PROGRAM MAIN
VAR



	SGO: TOGGLE;
	SGC: TOGGLE;
	TRU: TOGGLE;
	TRD: TOGGLE;
	VS: TOGGLE;
	TFS: TOGGLE;
	HSC: TOGGLE;
	HSO: TOGGLE;
	HDO: TOGGLE;
	HDC: TOGGLE;
	LC: TOGGLE;
	LR: TOGGLE;


	Eject_Empty_Pallet: BOOL;
	Empty_Pallet_Ejecting: BOOL;
	Empty_Pallet: BOOL;
	Full_Pallet: BOOL;
	Shroud_Latch: BOOL;


	Hoist_Cycle: BOOL;
	Next_Tier: BOOL;
	Hoist_Up_Disable: BOOL;
	ChainHoist_Enable: BOOL;
	Rev_Enable: BOOL;

	Auto_Tog: TOGGLE;



	Delay_Pallet_Advance2: TON;

	Delay_Pallet_Advance: TON;
	sChamberChain_Run: BOOL;
	Hoist_Down_Complete_TMR: TON;
	Discharge1_Pallet: BOOL;
	Eject_Cycle_TMR: TON;
	Hoist_Up_Tog: TOGGLE;
	Height_TMR: TOF;
	Reset_One_Shot: TP;
	sHoistUpDisable: BOOL;
	sChainHoistDn: BOOL;
	Fwd_Delay: TON;
	sCarriage_to_Pickup: BOOL;

	Open_Delay: TON;

	Release_Capture: TOF;
	DR2_Tog: TOGGLE;
	DR3_Tog: TOGGLE;
	DR4_Tog: TOGGLE;
	HoistUpDisableTog: TOGGLE;
	Gate_Closure_TMR:TON;




	Pa1Tog: TOGGLE;
	OpenTMR: TOF;
	CloseTMR: TOF;
	Down_Slow_Delay: TON;
	DSD: TIME;
	test: BOOL;
	Last_TierTMR1: TOF;
	Last_TierTMR2: TON;

	Down_Completion_TMR: TOF;
	Maintainloading: TOF;
	Ejecting_Pallet: BOOL;
	EmptyPallet_Jam_TMR: TON;





	TopFrameRem: TOF;
	Hoist_OneShot: TP;
	Hoist_Dn_Fast_Limit: TON;
	HDFL: TIME;
	Carriage_Disable_For_New_Pallet: BOOL;
	Slow_Reset: TP;
	LCT_Maintain: TOF;
	TT_Maintain: TOF;
	Disch1_Maintain: TOF;
	Disch2_Maintain: TOF;



	AutoLoadingTog: TOGGLE;
	ManualLoadingTog: TOGGLE;

	StopHoist_Tog: TOGGLE;

	TableTopJam: TON;
	Disch2Delay: TON;

	Discharge2Jam: TON;


	Disch2Full: TON;
	DR3TP: TP;
	Discharge2TOG: TOGGLE;
	Can_Count_M2: CTU;
	CC2: REAL;
	CanCount2A: CTU;
	CanCount2B: CTU;
	CC2B: REAL;
	CanCntReset: BOOL;
	CC2_Tens: REAL;

	FwdMaintain: TOF;
	Top_Frame_Removal: TON;
	Carriage_Forward_Enable: BOOL;
	Close_Pulse: TP;
	TT_Jam_Manager: TOF;
	Reverse_Delay: TON;
	Flash1_NP: TON;
	Flash2_NP: TOF;


	Flash1B: TON;
	Flash2B: TOF;
	mt: TOF;
	SlowTest: BOOL;
	Down_Slow_Maintain: TOF;
	Last_Slip_Sheet: TON;
	Test1: BOOL;
	Test2: BOOL;
	Empty_Pallet_Pulse: TP;
	Clank2_TMR: TON;
	Discharge_Run_TMR: TOF;
	Carriage_Slow_Enable: BOOL;
	Slow_Maintain: TOF;
	sc_DepalM2Count: INT;
	M2CanCounter2: CTU;
	M2CanCounter3: CTU;
	sc_Depal2Count3: BOOL;
	sc_Depal2Count2: BOOL;
	sc_Depal2Count13: INT;
	sc_Depal2Count12: INT;
	M2CanCounter4: CTU;
	M2CanCounter33: CTU;
	M2CanCounter34: CTU;
	a: INT;
	b: INT;
	C: INT;
	M2CanCounter333: CTU;
	d: INT;
	e: INT;
	F: INT;
	M2CanCounter333333: CTU;
	M: INT;
	DFS: CTU;
	LINCOLN: BOOL;

	LDS: BOOL;
	DSS: BOOL;
	K: INT;
	KJSJHE: BOOL;
	PLOP: INT;
	HLJKLTFK: CTU;
	FGHJD: INT;
	CancounterM2: CTU;
	CancounterM12: CTU;
	sc_Depal1_1stshiftcount: INT;
	try: INT;
	COUNTPULSE: BOOL;
	_TEST: CTU;
	_1stshiftcc: INT;
	_2NDshiftcc: INT;
	sc_M1CCReset: BOOL;
	Pallet_Count: INT;
	EmptyCans_Initial: REAL;
	InitialPalletCount: INT:=3276;
	TESTPALLETCOUNT: CTU;
	TESTPC: INT;
	M2CanCNTPE: BOOL;
	M2CanCountPE: BOOL;
	CanCounterCTU: CTU;
	CanCountWORD: WORD;
	CanCountMultiplier: CTU;
	MultiplierWORD: WORD;
	HighCount: REAL;
	MultiplierREAL: REAL;
	CanCountREAL: REAL;
	ActualCount: REAL;
	ChainHoistDown: Toggle;
	CHainHoistUp: TOGGLE;
	Infeed1: TOGGLE;
	ElevatorInfeed: TOGGLE;
	Elevatorrev: TOGGLE;
	Infeed2: Toggle;
	Infeed2REV: Toggle;
	Infeed1REV: TOGGLE;
	ELETOggle: TOGGLE;
	Cap: TOGGLE;
	Capture: TOGGLE;
	Release: TOGGLE;
	Rel: TOGGLE;
	hsclose: TOGGLE;
	sHoistSClose: BOOL;
	ABCD: TOGGLE;
	efgh: TOGGLE;
	CarFwd: Toggle;
	CarRev: Toggle;
	sDischarge1Run: BOOL;
	Discharge1Toggle: Toggle;
	Discharge2Run: Toggle;
	sDischarge2Run: BOOL;
	GD1: BOOL;
	Verify: TON;
	SetForNewPallet: SR;
	SendCarriageBack: BOOL;
	SetCarrRev: BOOL;
	Hoist_Tog_Resets: BOOL;
END_VAR
VAR_INPUT
	ProductHeight_Pos: BOOL;
	Carriage_to_Pickup: BOOL;
	Fwd_Enable: BOOL;
	DR1_Tog: TOGGLE;


END_VAR
VAR // added by the converter: edge detectors and wires of the graphical bodies
    _w1, _w2, _w3, _w4, _w5, _w6, _w7, _w8 : BOOL;
END_VAR

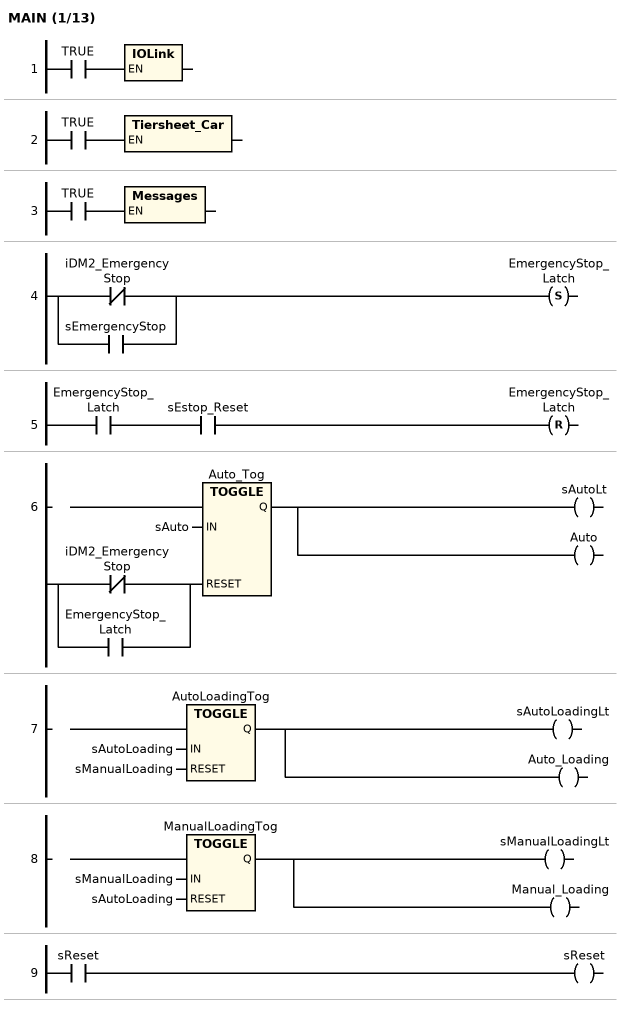
// NETWORK 1
IOLink();

// NETWORK 2
Tiersheet_Car();

// NETWORK 3
Messages();

// NETWORK 4
EmergencyStop_Latch S= NOT iDM2_EmergencyStop OR sEmergencyStop;

// NETWORK 5
EmergencyStop_Latch R= EmergencyStop_Latch AND sEstop_Reset;

// NETWORK 6
Auto_Tog(IN := sAuto, RESET := NOT iDM2_EmergencyStop OR EmergencyStop_Latch); // TOGGLE
sAutoLt := Auto_Tog.Q;
Auto := Auto_Tog.Q;

// NETWORK 7
AutoLoadingTog(IN := sAutoLoading, RESET := sManualLoading); // TOGGLE
sAutoLoadingLt := AutoLoadingTog.Q;
Auto_Loading := AutoLoadingTog.Q;

// NETWORK 8
ManualLoadingTog(IN := sManualLoading, RESET := sAutoLoading); // TOGGLE
sManualLoadingLt := ManualLoadingTog.Q;
Manual_Loading := ManualLoadingTog.Q;

// NETWORK 9
sReset := sReset;

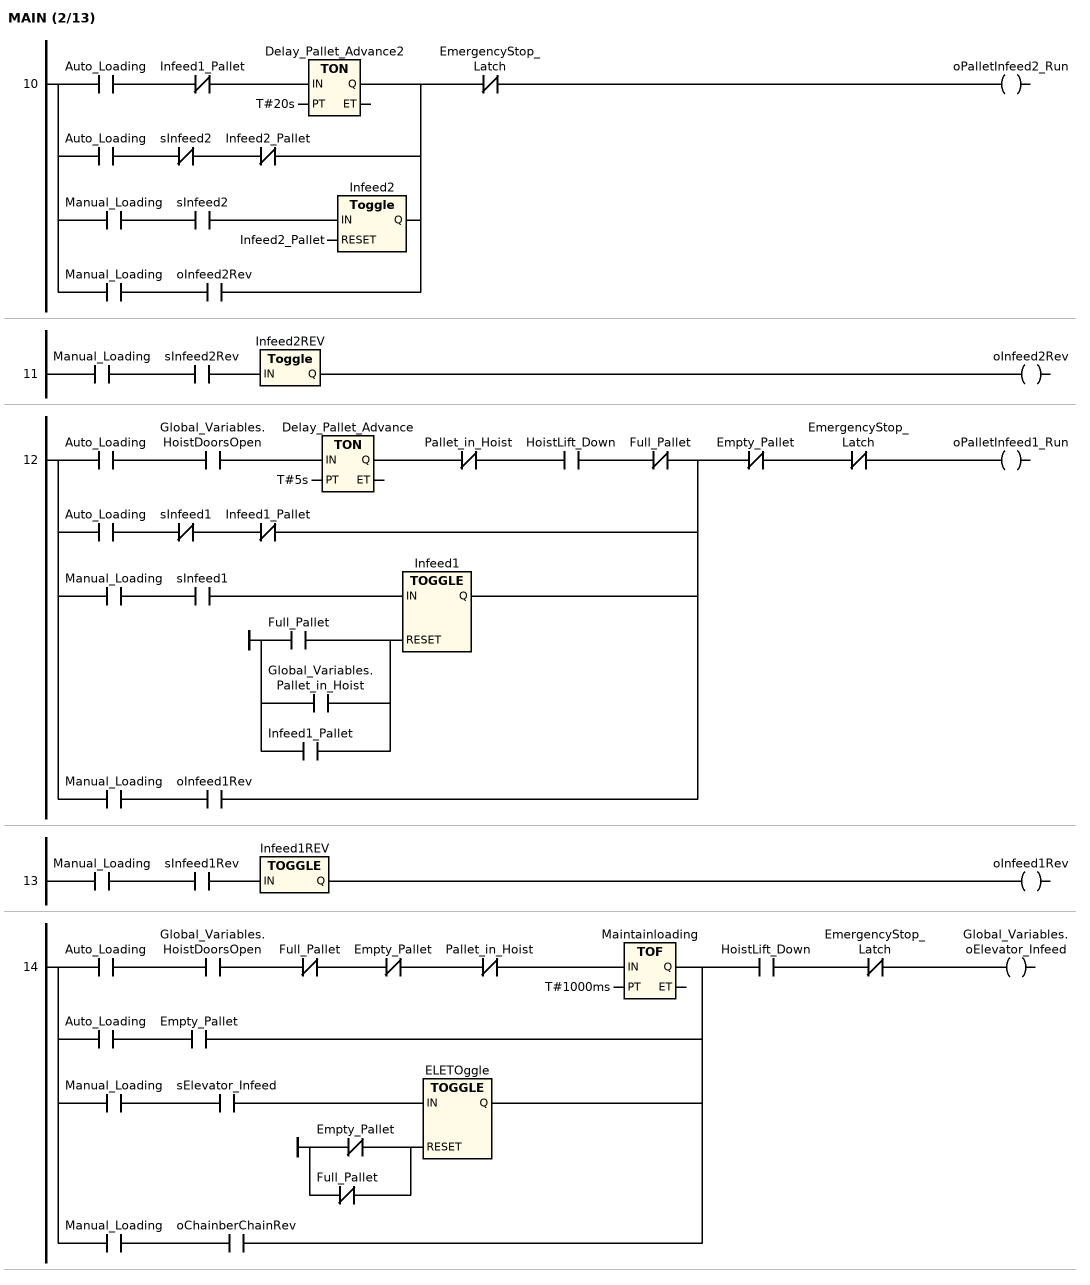
// NETWORK 10
Delay_Pallet_Advance2(IN := Auto_Loading AND NOT Infeed1_Pallet, PT := T#20s); // TON
Infeed2(IN := Manual_Loading AND sInfeed2, RESET := Infeed2_Pallet); // Toggle
oPalletInfeed2_Run := (Delay_Pallet_Advance2.Q OR Auto_Loading AND NOT sInfeed2 AND NOT Infeed2_Pallet OR Infeed2.Q OR Manual_Loading AND oInfeed2Rev) AND NOT EmergencyStop_Latch;

// NETWORK 11
Infeed2REV(IN := Manual_Loading AND sInfeed2Rev); // Toggle
oInfeed2Rev := Infeed2REV.Q;

// NETWORK 12
Delay_Pallet_Advance(IN := Auto_Loading AND Global_Variables.HoistDoorsOpen, PT := T#5s); // TON
Infeed1(IN := Manual_Loading AND sInfeed1, RESET := Full_Pallet OR Global_Variables.Pallet_in_Hoist OR Infeed1_Pallet); // TOGGLE
oPalletInfeed1_Run := (Delay_Pallet_Advance.Q AND NOT Pallet_in_Hoist AND HoistLift_Down AND NOT Full_Pallet OR Auto_Loading AND NOT sInfeed1 AND NOT Infeed1_Pallet OR Infeed1.Q OR Manual_Loading AND oInfeed1Rev) AND NOT Empty_Pallet AND NOT EmergencyStop_Latch;

// NETWORK 13
Infeed1REV(IN := Manual_Loading AND sInfeed1Rev); // TOGGLE
oInfeed1Rev := Infeed1REV.Q;

// NETWORK 14
Maintainloading(IN := Auto_Loading AND Global_Variables.HoistDoorsOpen AND NOT Full_Pallet AND NOT Empty_Pallet AND NOT Pallet_in_Hoist, PT := T#1000ms); // TOF
ELETOggle(IN := Manual_Loading AND sElevator_Infeed, RESET := NOT Empty_Pallet OR NOT Full_Pallet); // TOGGLE
Global_Variables.oElevator_Infeed := (Maintainloading.Q OR Auto_Loading AND Empty_Pallet OR ELETOggle.Q OR Manual_Loading AND oChainberChainRev) AND HoistLift_Down AND NOT EmergencyStop_Latch;

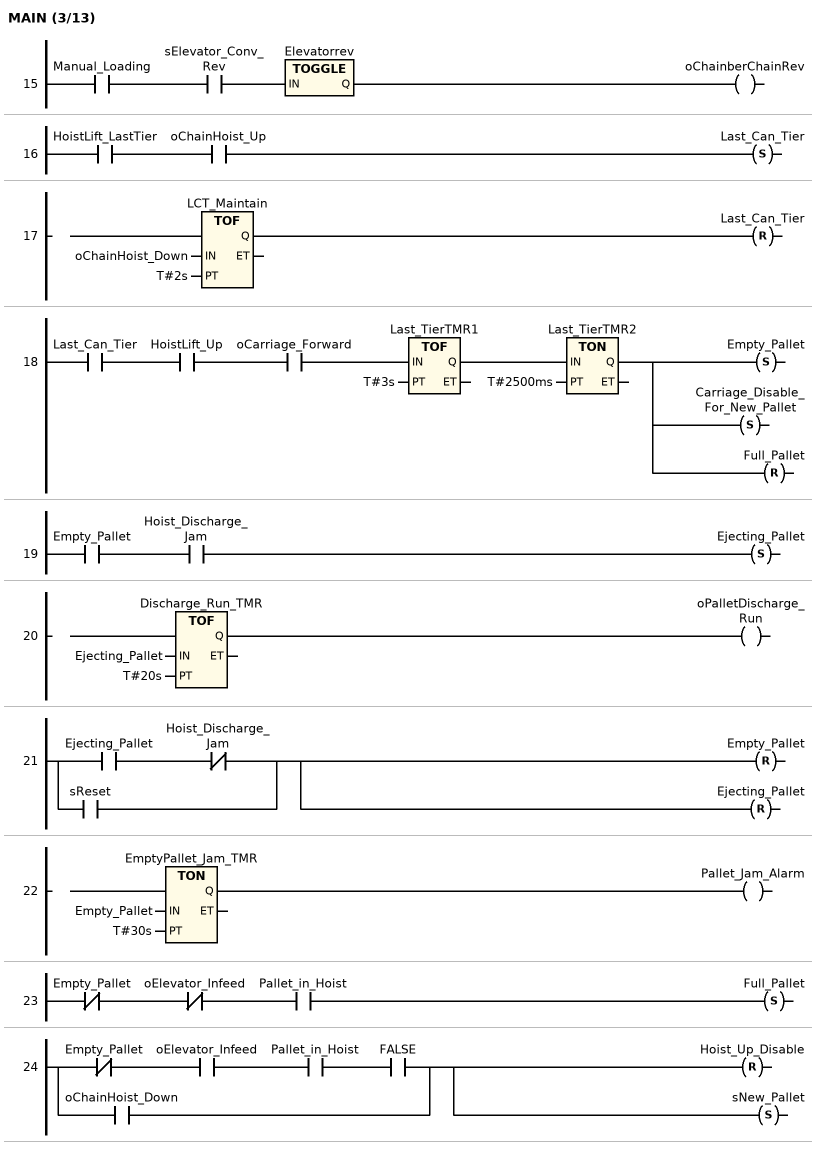
// NETWORK 15
Elevatorrev(IN := Manual_Loading AND sElevator_Conv_Rev); // TOGGLE
oChainberChainRev := Elevatorrev.Q;

// NETWORK 16
Last_Can_Tier S= HoistLift_LastTier AND oChainHoist_Up;

// NETWORK 17
LCT_Maintain(IN := oChainHoist_Down, PT := T#2s); // TOF
Last_Can_Tier R= LCT_Maintain.Q;

// NETWORK 18
Last_TierTMR1(IN := Last_Can_Tier AND HoistLift_Up AND oCarriage_Forward, PT := T#3s); // TOF
Last_TierTMR2(IN := Last_TierTMR1.Q, PT := T#2500ms); // TON
Empty_Pallet S= Last_TierTMR2.Q;
Carriage_Disable_For_New_Pallet S= Last_TierTMR2.Q;
Full_Pallet R= Last_TierTMR2.Q;

// NETWORK 19
Ejecting_Pallet S= Empty_Pallet AND Hoist_Discharge_Jam;

// NETWORK 20
Discharge_Run_TMR(IN := Ejecting_Pallet, PT := T#20s); // TOF
oPalletDischarge_Run := Discharge_Run_TMR.Q;

// NETWORK 21
_w1 := Ejecting_Pallet AND NOT Hoist_Discharge_Jam OR sReset;
Empty_Pallet R= _w1;
Ejecting_Pallet R= _w1;

// NETWORK 22
EmptyPallet_Jam_TMR(IN := Empty_Pallet, PT := T#30s); // TON
Pallet_Jam_Alarm := EmptyPallet_Jam_TMR.Q;

// NETWORK 23
Full_Pallet S= NOT Empty_Pallet AND NOT oElevator_Infeed AND Pallet_in_Hoist;

// NETWORK 24
_w2 := NOT Empty_Pallet AND oElevator_Infeed AND Pallet_in_Hoist AND FALSE OR oChainHoist_Down;
Hoist_Up_Disable R= _w2;
sNew_Pallet S= _w2;

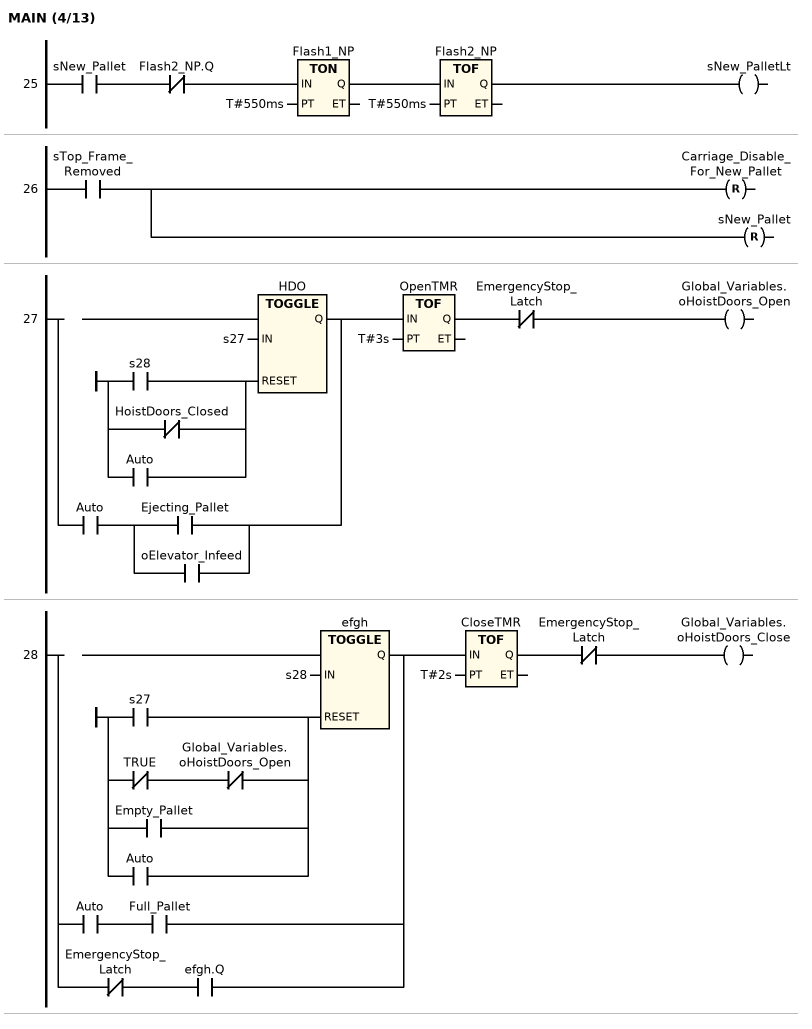
// NETWORK 25
Flash1_NP(IN := sNew_Pallet AND NOT Flash2_NP.Q, PT := T#550ms); // TON
Flash2_NP(IN := Flash1_NP.Q, PT := T#550ms); // TOF
sNew_PalletLt := Flash2_NP.Q;

// NETWORK 26
Carriage_Disable_For_New_Pallet R= sTop_Frame_Removed;
sNew_Pallet R= sTop_Frame_Removed;

// NETWORK 27
HDO(IN := s27, RESET := s28 OR NOT HoistDoors_Closed OR Auto); // TOGGLE
OpenTMR(IN := HDO.Q OR Auto AND (Ejecting_Pallet OR oElevator_Infeed), PT := T#3s); // TOF
Global_Variables.oHoistDoors_Open := OpenTMR.Q AND NOT EmergencyStop_Latch;

// NETWORK 28
efgh(IN := s28, RESET := s27 OR NOT TRUE AND NOT Global_Variables.oHoistDoors_Open OR Empty_Pallet OR Auto); // TOGGLE
CloseTMR(IN := efgh.Q OR Auto AND Full_Pallet OR NOT EmergencyStop_Latch AND efgh.Q, PT := T#2s); // TOF
Global_Variables.oHoistDoors_Close := CloseTMR.Q AND NOT EmergencyStop_Latch;

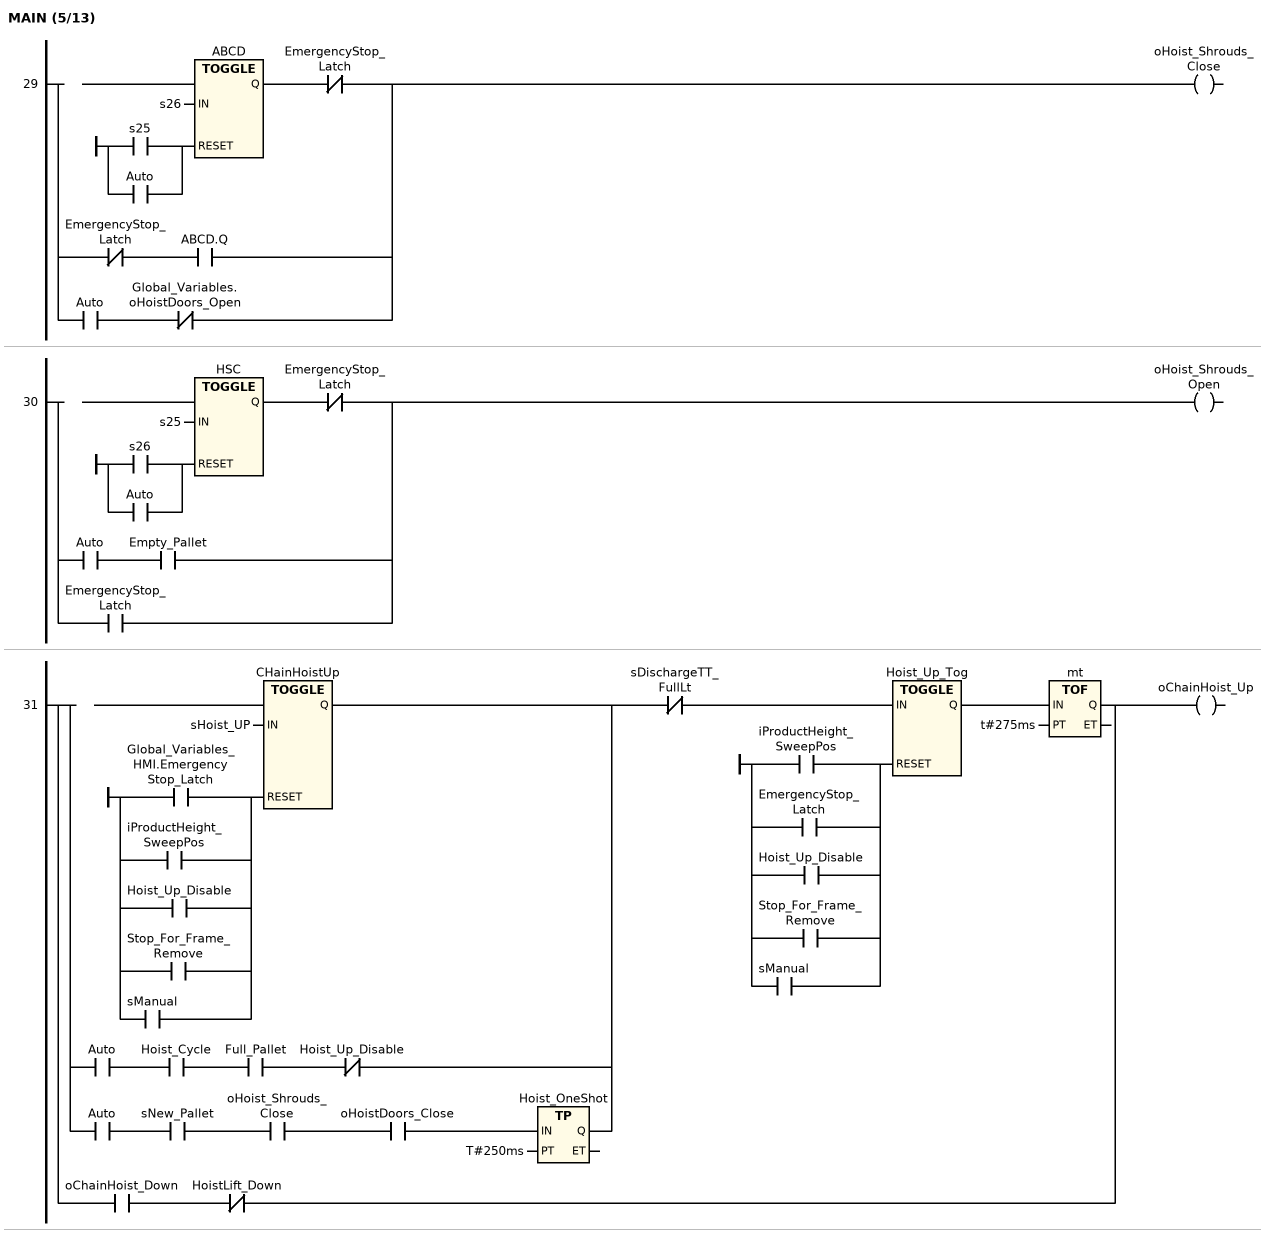
// NETWORK 29
ABCD(IN := s26, RESET := s25 OR Auto); // TOGGLE
oHoist_Shrouds_Close := ABCD.Q AND NOT EmergencyStop_Latch OR NOT EmergencyStop_Latch AND ABCD.Q OR Auto AND NOT Global_Variables.oHoistDoors_Open;

// NETWORK 30
HSC(IN := s25, RESET := s26 OR Auto); // TOGGLE
oHoist_Shrouds_Open := HSC.Q AND NOT EmergencyStop_Latch OR Auto AND Empty_Pallet OR EmergencyStop_Latch;

// NETWORK 31
CHainHoistUp(IN := sHoist_UP, RESET := Global_Variables_HMI.EmergencyStop_Latch OR iProductHeight_SweepPos OR Hoist_Up_Disable OR Stop_For_Frame_Remove OR sManual); // TOGGLE
Hoist_OneShot(IN := Auto AND sNew_Pallet AND oHoist_Shrouds_Close AND oHoistDoors_Close, PT := T#250ms); // TP
Hoist_Up_Tog(IN := (CHainHoistUp.Q OR Auto AND Hoist_Cycle AND Full_Pallet AND NOT Hoist_Up_Disable OR Hoist_OneShot.Q) AND NOT sDischargeTT_FullLt, RESET := iProductHeight_SweepPos OR EmergencyStop_Latch OR Hoist_Up_Disable OR Stop_For_Frame_Remove OR sManual); // TOGGLE
mt(IN := Hoist_Up_Tog.Q, PT := t#275ms); // TOF
oChainHoist_Up := mt.Q OR oChainHoist_Down AND NOT HoistLift_Down;

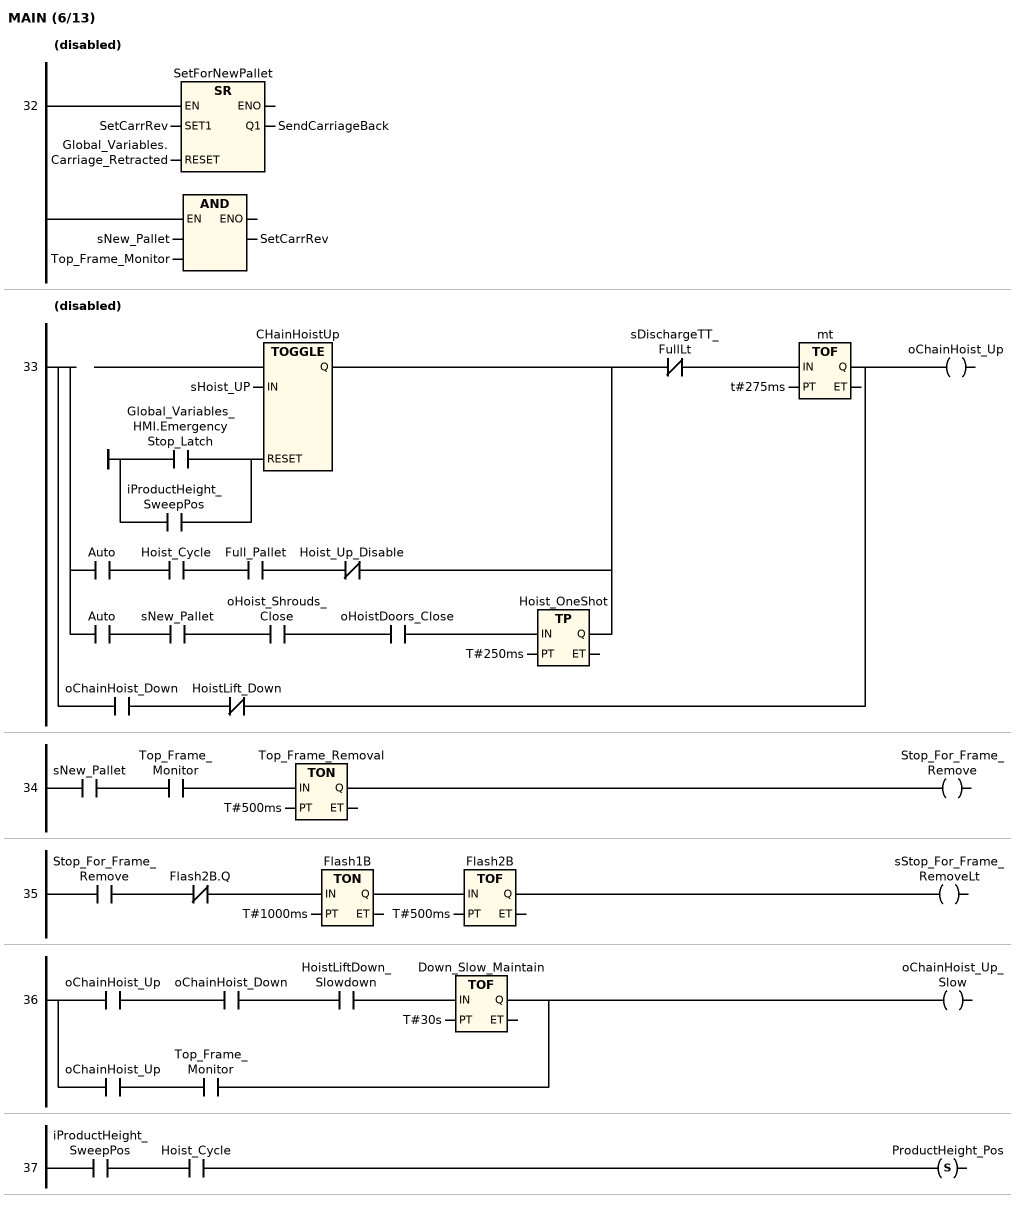
// NETWORK 32 (disabled)
// SetForNewPallet(SET1 := SetCarrRev, RESET := Global_Variables.Carriage_Retracted, Q1 => SendCarriageBack); // SR
// SetCarrRev := sNew_Pallet AND Top_Frame_Monitor;

// NETWORK 33 (disabled)
// CHainHoistUp(IN := sHoist_UP, RESET := Global_Variables_HMI.EmergencyStop_Latch OR iProductHeight_SweepPos); // TOGGLE
// Hoist_OneShot(IN := Auto AND sNew_Pallet AND oHoist_Shrouds_Close AND oHoistDoors_Close, PT := T#250ms); // TP
// mt(IN := (CHainHoistUp.Q OR Auto AND Hoist_Cycle AND Full_Pallet AND NOT Hoist_Up_Disable OR Hoist_OneShot.Q) AND NOT sDischargeTT_FullLt, PT := t#275ms); // TOF
// oChainHoist_Up := mt.Q OR oChainHoist_Down AND NOT HoistLift_Down;

// NETWORK 34
Top_Frame_Removal(IN := sNew_Pallet AND Top_Frame_Monitor, PT := T#500ms); // TON
Stop_For_Frame_Remove := Top_Frame_Removal.Q;

// NETWORK 35
Flash1B(IN := Stop_For_Frame_Remove AND NOT Flash2B.Q, PT := T#1000ms); // TON
Flash2B(IN := Flash1B.Q, PT := T#500ms); // TOF
sStop_For_Frame_RemoveLt := Flash2B.Q;

// NETWORK 36
Down_Slow_Maintain(IN := oChainHoist_Up AND (oChainHoist_Down AND HoistLiftDown_Slowdown), PT := T#30s); // TOF
oChainHoist_Up_Slow := Down_Slow_Maintain.Q OR oChainHoist_Up AND Top_Frame_Monitor;

// NETWORK 37
ProductHeight_Pos S= iProductHeight_SweepPos AND Hoist_Cycle;

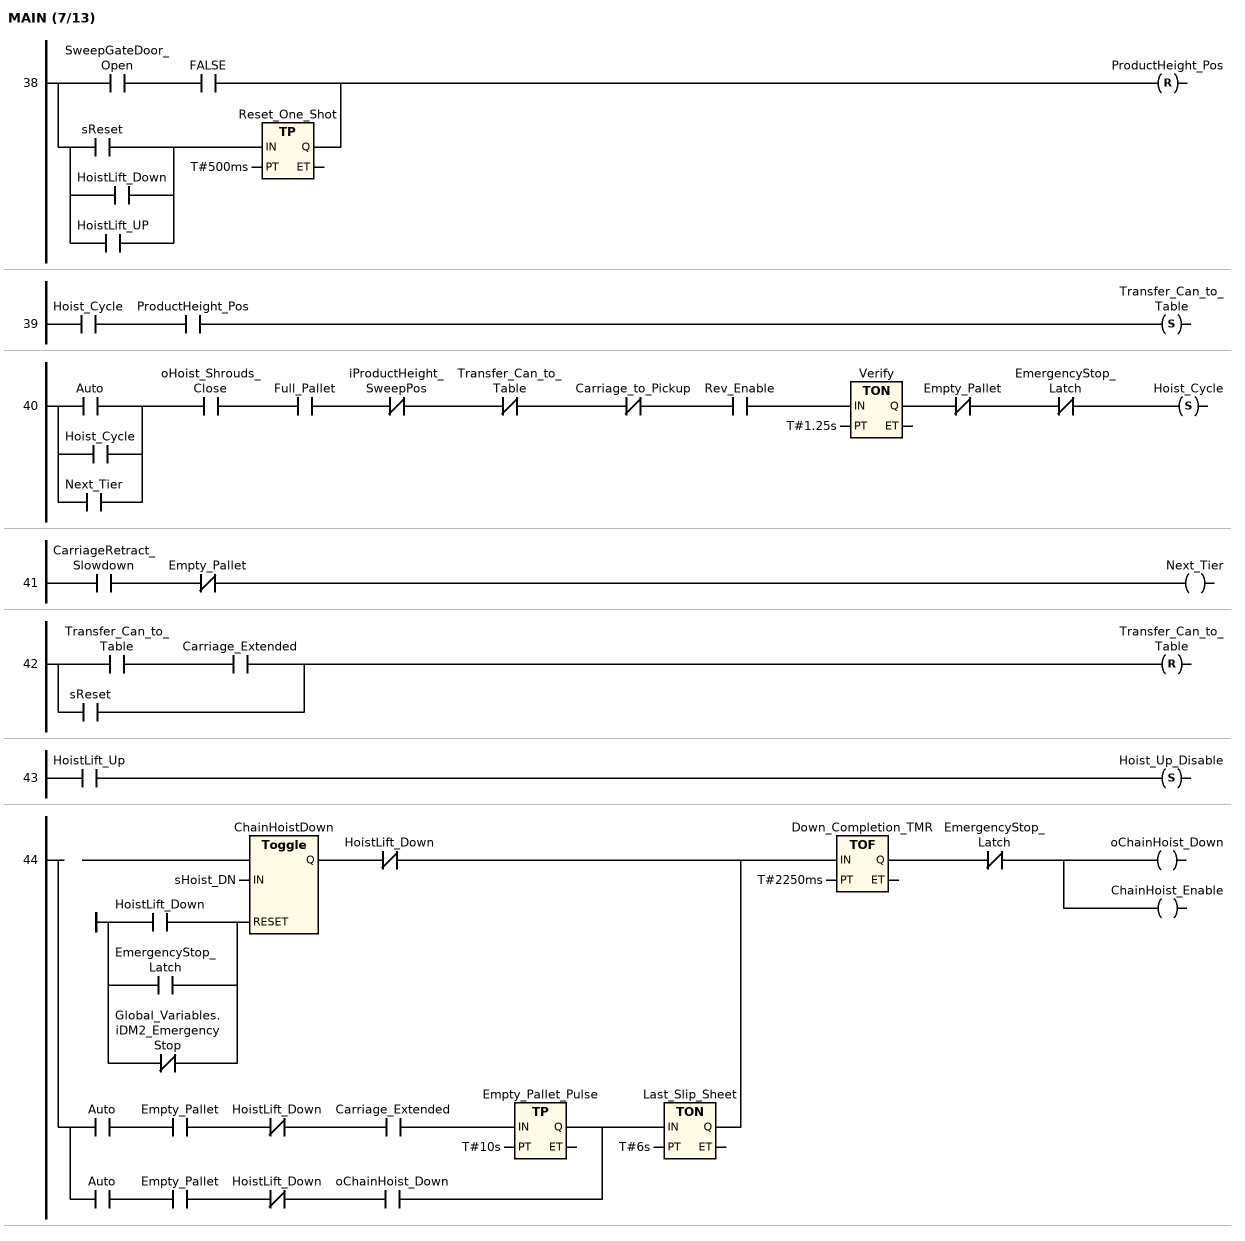
// NETWORK 38
Reset_One_Shot(IN := sReset OR HoistLift_Down OR HoistLift_UP, PT := T#500ms); // TP
ProductHeight_Pos R= SweepGateDoor_Open AND FALSE OR Reset_One_Shot.Q;

// NETWORK 39
Transfer_Can_to_Table S= Hoist_Cycle AND ProductHeight_Pos;

// NETWORK 40
Verify(IN := (Auto OR Hoist_Cycle OR Next_Tier) AND oHoist_Shrouds_Close AND Full_Pallet AND NOT iProductHeight_SweepPos AND NOT Transfer_Can_to_Table AND NOT Carriage_to_Pickup AND Rev_Enable, PT := T#1.25s); // TON
Hoist_Cycle S= Verify.Q AND NOT Empty_Pallet AND NOT EmergencyStop_Latch;

// NETWORK 41
Next_Tier := CarriageRetract_Slowdown AND NOT Empty_Pallet;

// NETWORK 42
Transfer_Can_to_Table R= Transfer_Can_to_Table AND Carriage_Extended OR sReset;

// NETWORK 43
Hoist_Up_Disable S= HoistLift_Up;

// NETWORK 44
ChainHoistDown(IN := sHoist_DN, RESET := HoistLift_Down OR EmergencyStop_Latch OR NOT Global_Variables.iDM2_EmergencyStop); // Toggle
Empty_Pallet_Pulse(IN := Auto AND Empty_Pallet AND NOT HoistLift_Down AND Carriage_Extended, PT := T#10s); // TP
Last_Slip_Sheet(IN := Empty_Pallet_Pulse.Q OR Auto AND Empty_Pallet AND NOT HoistLift_Down AND oChainHoist_Down, PT := T#6s); // TON
Down_Completion_TMR(IN := ChainHoistDown.Q AND NOT HoistLift_Down OR Last_Slip_Sheet.Q, PT := T#2250ms); // TOF
_w3 := Down_Completion_TMR.Q AND NOT EmergencyStop_Latch;
oChainHoist_Down := _w3;
ChainHoist_Enable := _w3;

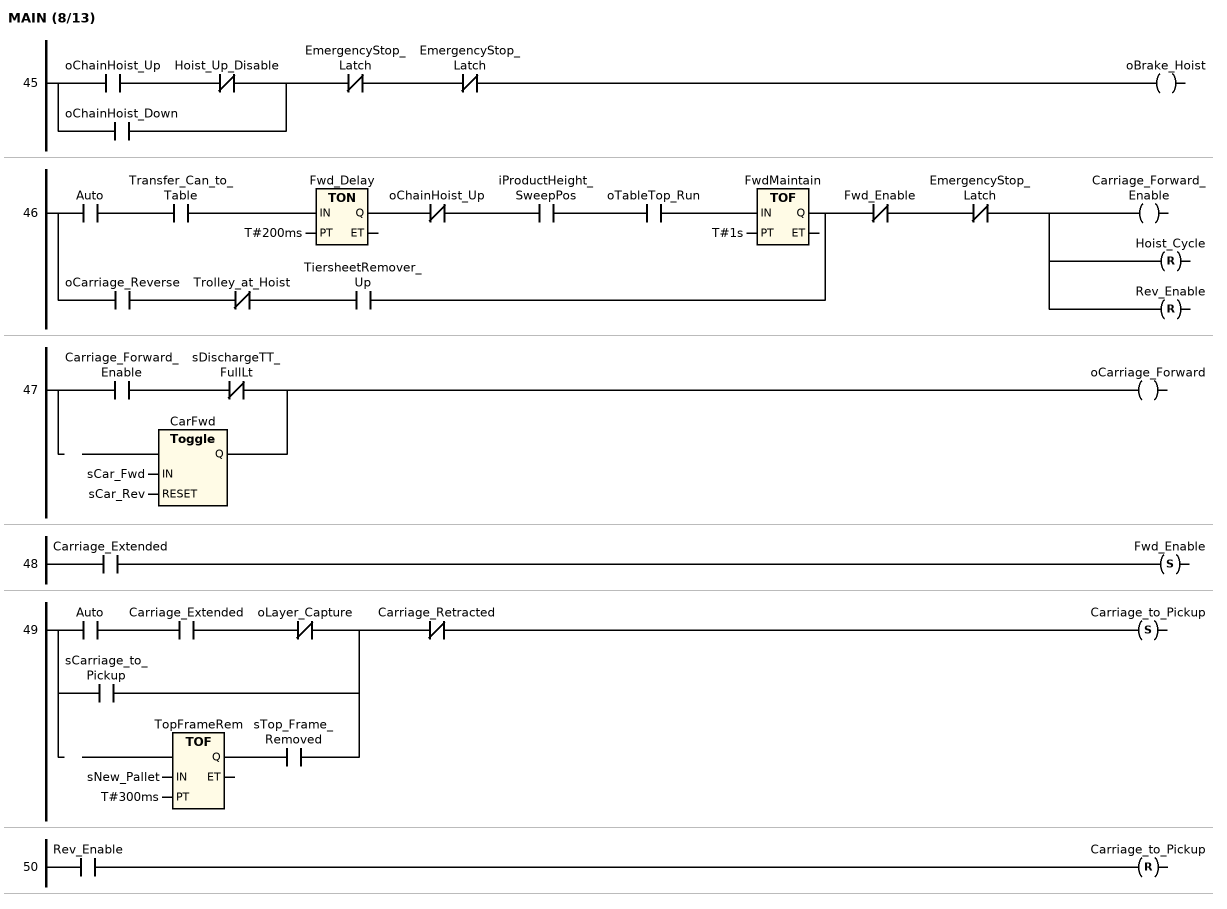
// NETWORK 45
oBrake_Hoist := (oChainHoist_Up AND NOT Hoist_Up_Disable OR oChainHoist_Down) AND NOT EmergencyStop_Latch AND NOT EmergencyStop_Latch;

// NETWORK 46
Fwd_Delay(IN := Auto AND Transfer_Can_to_Table, PT := T#200ms); // TON
FwdMaintain(IN := Fwd_Delay.Q AND NOT oChainHoist_Up AND iProductHeight_SweepPos AND oTableTop_Run, PT := T#1s); // TOF
_w4 := (FwdMaintain.Q OR oCarriage_Reverse AND NOT Trolley_at_Hoist AND TiersheetRemover_Up) AND NOT Fwd_Enable AND NOT EmergencyStop_Latch;
Carriage_Forward_Enable := _w4;
Hoist_Cycle R= _w4;
Rev_Enable R= _w4;

// NETWORK 47
CarFwd(IN := sCar_Fwd, RESET := sCar_Rev); // Toggle
oCarriage_Forward := Carriage_Forward_Enable AND NOT sDischargeTT_FullLt OR CarFwd.Q;

// NETWORK 48
Fwd_Enable S= Carriage_Extended;

// NETWORK 49
TopFrameRem(IN := sNew_Pallet, PT := T#300ms); // TOF
Carriage_to_Pickup S= (Auto AND Carriage_Extended AND NOT oLayer_Capture OR sCarriage_to_Pickup OR TopFrameRem.Q AND sTop_Frame_Removed) AND NOT Carriage_Retracted;

// NETWORK 50
Carriage_to_Pickup R= Rev_Enable;

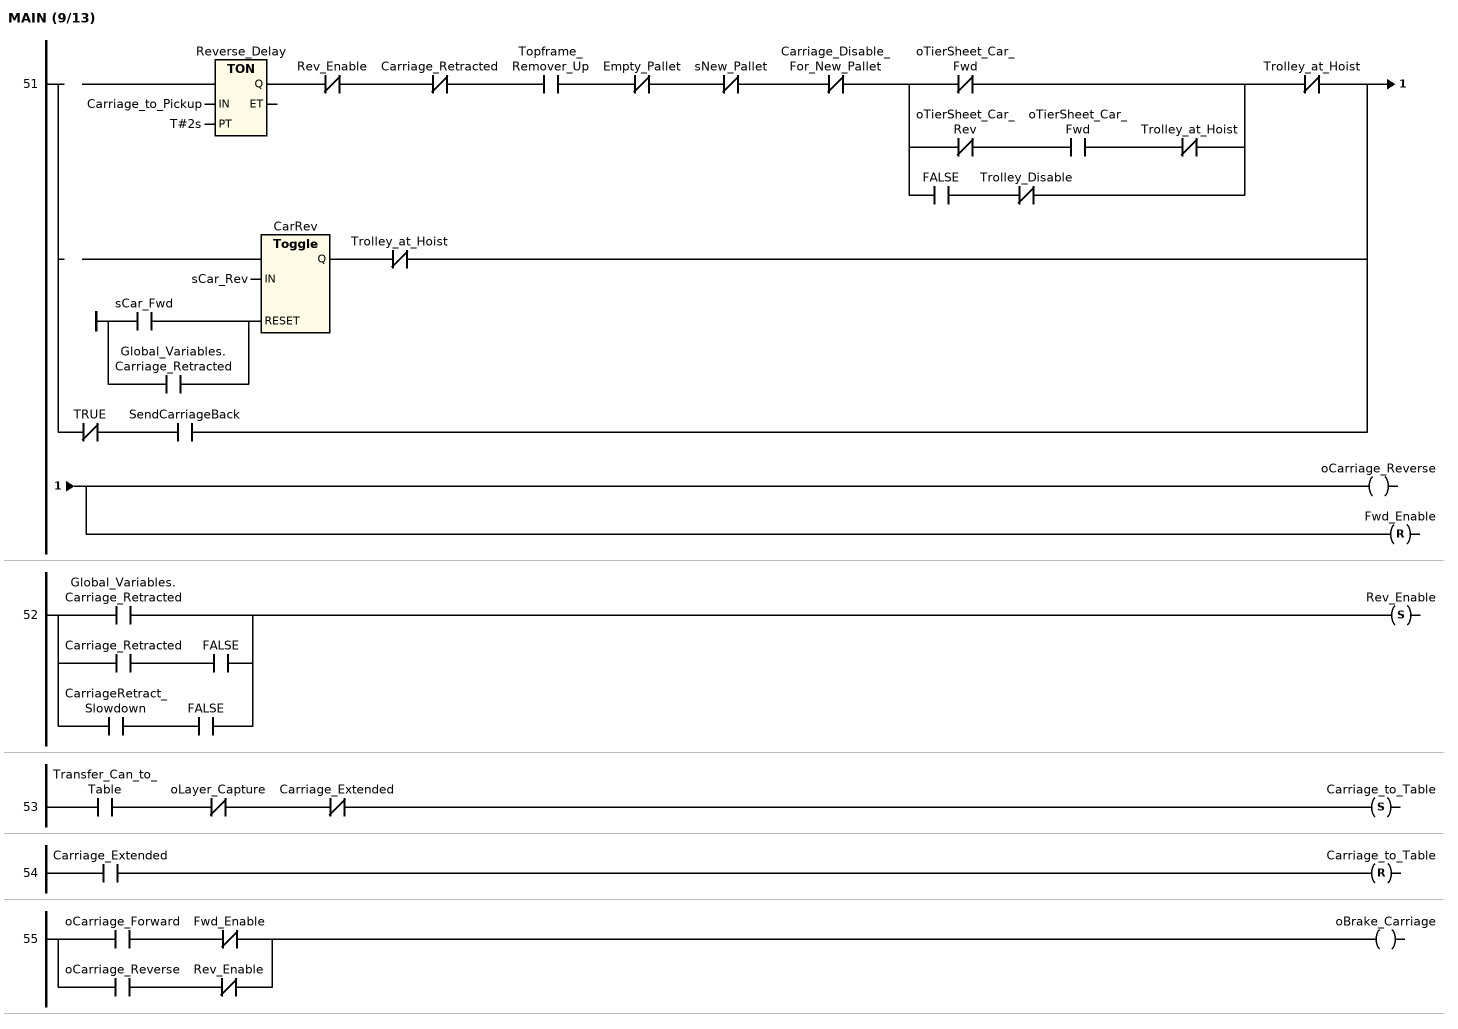
// NETWORK 51
Reverse_Delay(IN := Carriage_to_Pickup, PT := T#2s); // TON
CarRev(IN := sCar_Rev, RESET := sCar_Fwd OR Global_Variables.Carriage_Retracted); // Toggle
_w5 := Reverse_Delay.Q AND NOT Rev_Enable AND NOT Carriage_Retracted AND Topframe_Remover_Up AND NOT Empty_Pallet AND NOT sNew_Pallet AND NOT Carriage_Disable_For_New_Pallet AND (NOT oTierSheet_Car_Fwd OR NOT oTierSheet_Car_Rev AND oTierSheet_Car_Fwd AND NOT Trolley_at_Hoist OR FALSE AND NOT Trolley_Disable) AND NOT Trolley_at_Hoist OR CarRev.Q AND NOT Trolley_at_Hoist OR NOT TRUE AND SendCarriageBack;
oCarriage_Reverse := _w5;
Fwd_Enable R= _w5;

// NETWORK 52
Rev_Enable S= Global_Variables.Carriage_Retracted OR Carriage_Retracted AND FALSE OR CarriageRetract_Slowdown AND FALSE;

// NETWORK 53
Carriage_to_Table S= Transfer_Can_to_Table AND NOT oLayer_Capture AND NOT Carriage_Extended;

// NETWORK 54
Carriage_to_Table R= Carriage_Extended;

// NETWORK 55
oBrake_Carriage := oCarriage_Forward AND NOT Fwd_Enable OR oCarriage_Reverse AND NOT Rev_Enable;

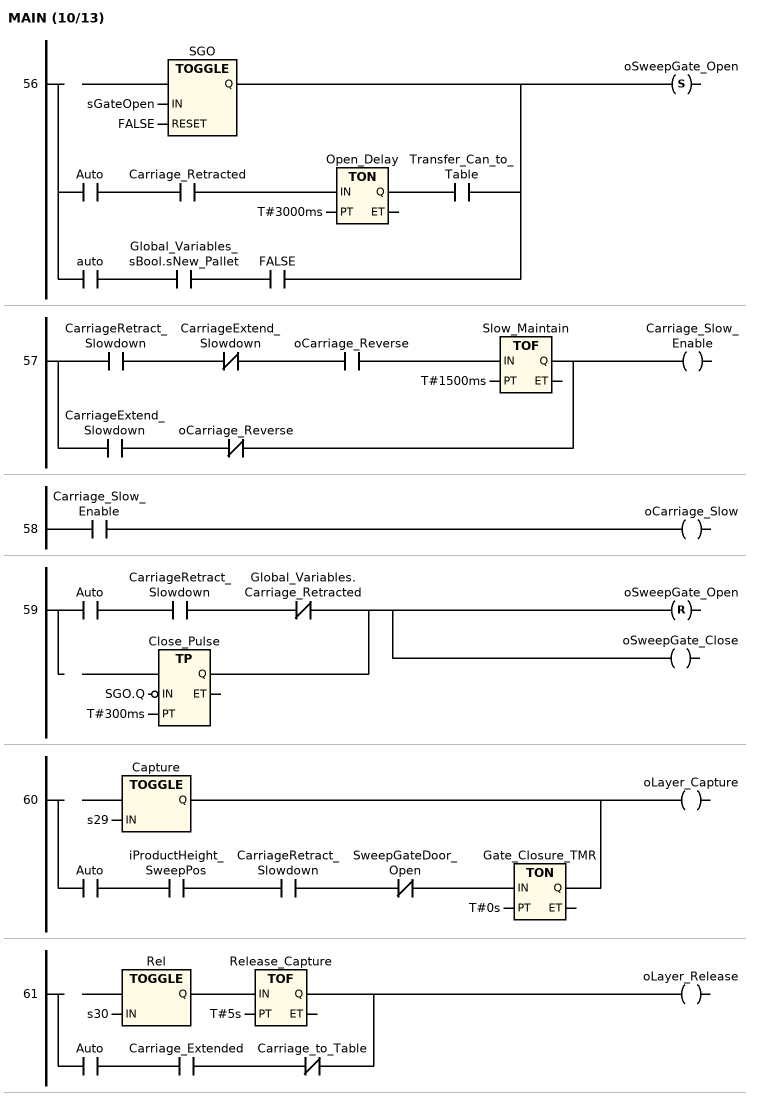
// NETWORK 56
SGO(IN := sGateOpen, RESET := FALSE); // TOGGLE
Open_Delay(IN := Auto AND Carriage_Retracted, PT := T#3000ms); // TON
oSweepGate_Open S= SGO.Q OR Open_Delay.Q AND Transfer_Can_to_Table OR auto AND Global_Variables_sBool.sNew_Pallet AND FALSE;

// NETWORK 57
Slow_Maintain(IN := CarriageRetract_Slowdown AND NOT CarriageExtend_Slowdown AND oCarriage_Reverse, PT := T#1500ms); // TOF
Carriage_Slow_Enable := Slow_Maintain.Q OR CarriageExtend_Slowdown AND NOT oCarriage_Reverse;

// NETWORK 58
oCarriage_Slow := Carriage_Slow_Enable;

// NETWORK 59
Close_Pulse(IN := NOT SGO.Q, PT := T#300ms); // TP
_w6 := Auto AND CarriageRetract_Slowdown AND NOT Global_Variables.Carriage_Retracted OR Close_Pulse.Q;
oSweepGate_Open R= _w6;
oSweepGate_Close := _w6;

// NETWORK 60
Capture(IN := s29); // TOGGLE
Gate_Closure_TMR(IN := Auto AND iProductHeight_SweepPos AND CarriageRetract_Slowdown AND NOT SweepGateDoor_Open, PT := T#0s); // TON
oLayer_Capture := Capture.Q OR Gate_Closure_TMR.Q;

// NETWORK 61
Rel(IN := s30); // TOGGLE
Release_Capture(IN := Rel.Q, PT := T#5s); // TOF
oLayer_Release := Release_Capture.Q OR Auto AND Carriage_Extended AND NOT Carriage_to_Table;

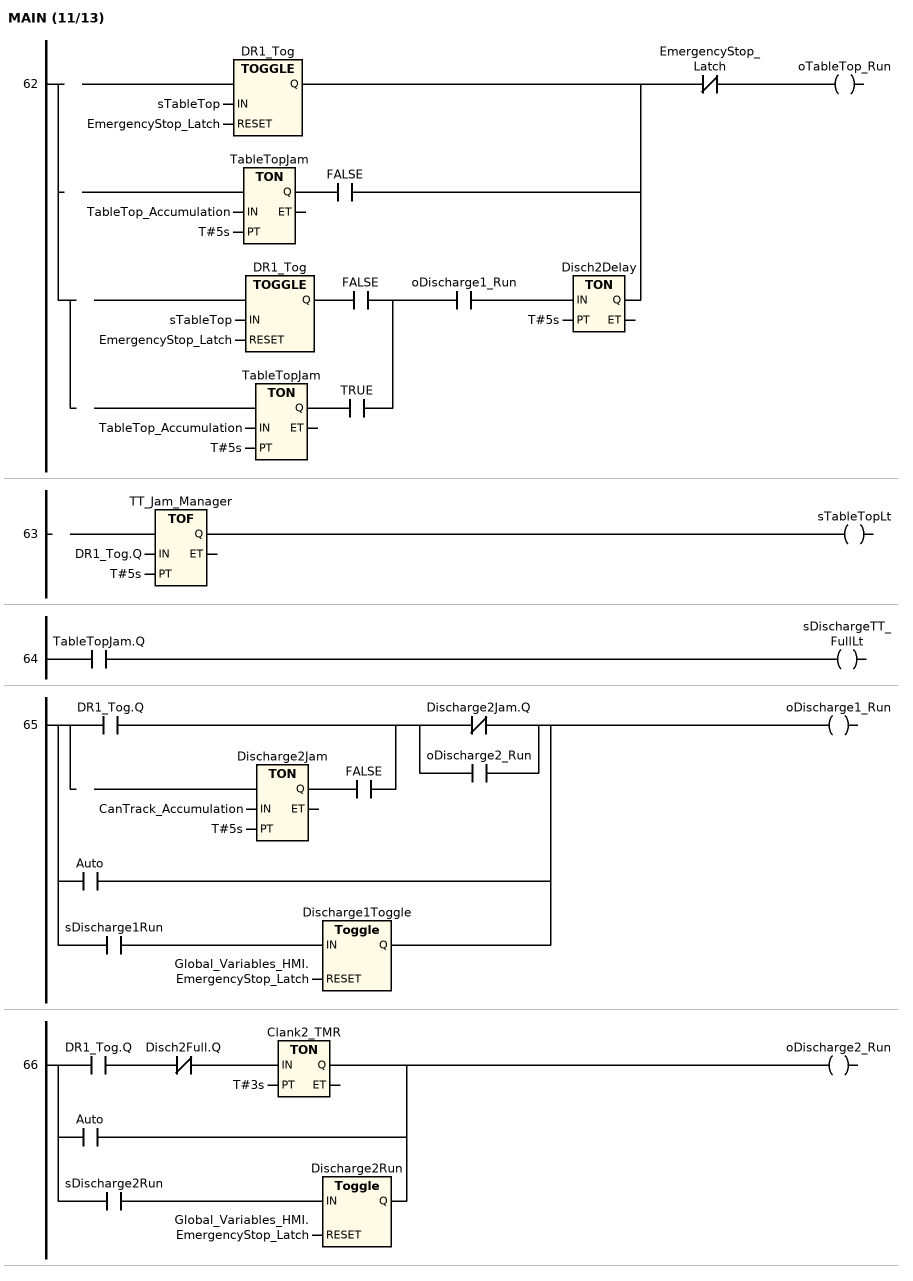
// NETWORK 62
DR1_Tog(IN := sTableTop, RESET := EmergencyStop_Latch); // TOGGLE
_w8 := DR1_Tog.Q;
TableTopJam(IN := TableTop_Accumulation, PT := T#5s); // TON
_w7 := TableTopJam.Q AND FALSE;
DR1_Tog(IN := sTableTop, RESET := EmergencyStop_Latch); // TOGGLE
TableTopJam(IN := TableTop_Accumulation, PT := T#5s); // TON
Disch2Delay(IN := (DR1_Tog.Q AND FALSE OR TableTopJam.Q AND TRUE) AND oDischarge1_Run, PT := T#5s); // TON
oTableTop_Run := (_w8 OR _w7 OR Disch2Delay.Q) AND NOT EmergencyStop_Latch;

// NETWORK 63
TT_Jam_Manager(IN := DR1_Tog.Q, PT := T#5s); // TOF
sTableTopLt := TT_Jam_Manager.Q;

// NETWORK 64
sDischargeTT_FullLt := TableTopJam.Q;

// NETWORK 65
Discharge2Jam(IN := CanTrack_Accumulation, PT := T#5s); // TON
Discharge1Toggle(IN := sDischarge1Run, RESET := Global_Variables_HMI.EmergencyStop_Latch); // Toggle
oDischarge1_Run := (DR1_Tog.Q OR Discharge2Jam.Q AND FALSE) AND (NOT Discharge2Jam.Q OR oDischarge2_Run) OR Auto OR Discharge1Toggle.Q;

// NETWORK 66
Clank2_TMR(IN := DR1_Tog.Q AND NOT Disch2Full.Q, PT := T#3s); // TON
Discharge2Run(IN := sDischarge2Run, RESET := Global_Variables_HMI.EmergencyStop_Latch); // Toggle
oDischarge2_Run := Clank2_TMR.Q OR Auto OR Discharge2Run.Q;

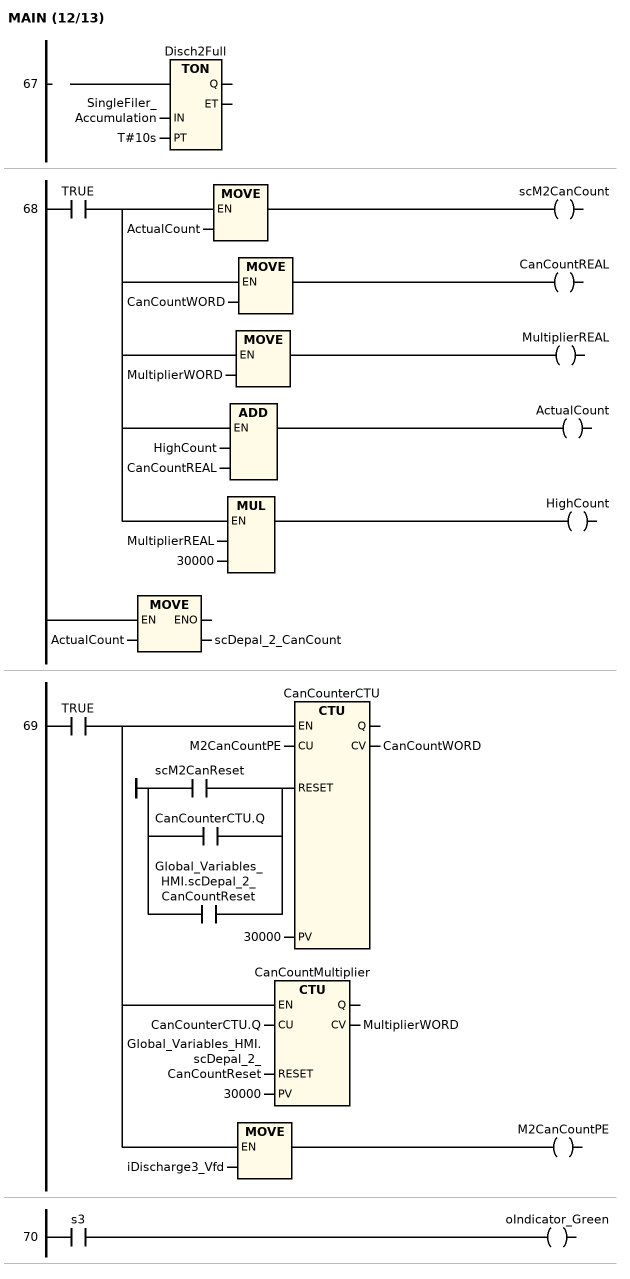
// NETWORK 67
Disch2Full(IN := SingleFiler_Accumulation, PT := T#10s); // TON

// NETWORK 68
scM2CanCount := ActualCount;
CanCountREAL := CanCountWORD;
MultiplierREAL := MultiplierWORD;
ActualCount := HighCount + CanCountREAL;
HighCount := MultiplierREAL * 30000;
scDepal_2_CanCount := ActualCount;

// NETWORK 69
CanCounterCTU(
    CU := M2CanCountPE,
    RESET := scM2CanReset OR CanCounterCTU.Q OR Global_Variables_HMI.scDepal_2_CanCountReset,
    PV := 30000,
    CV => CanCountWORD); // CTU
CanCountMultiplier(
    CU := CanCounterCTU.Q,
    RESET := Global_Variables_HMI.scDepal_2_CanCountReset,
    PV := 30000,
    CV => MultiplierWORD); // CTU
M2CanCountPE := iDischarge3_Vfd;

// NETWORK 70
oIndicator_Green := s3;

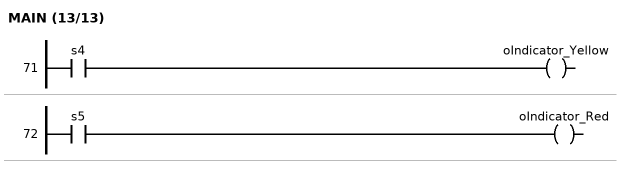
// NETWORK 71
oIndicator_Yellow := s4;

// NETWORK 72
oIndicator_Red := s5;

END_PROGRAM

(* stored: Version 1.1.0.1, ProductVersion 3.1.4024.15
   POU MAIN: Id {e81ee7b4-2f88-4f4f-8fbd-5aa9f13d476b}, SpecialFunc None *)
